// TIA Portal V20 export
TYPE "LKinCtrl_typePointCoordinates_PreBuf"
   STRUCT
      startPosition : Array[1..6] of LReal;   // absolute start position
      targetPosition : Array[1..6] of LReal;   // end position or relative distance depending on command type
      targetDistance : Array[1..6] of LReal;
      coordSystem : DInt := 0;   // 0: WCS; 1: OCS[1]; 2: OCS[2]; 3: OCS[3]
   END_STRUCT;
END_TYPE
